RESOURCE_TYPE _Core3
  (* Standard: 61499-2 *)
  (* Version 0.1, 2017-00-16, hpea485, UOA *)
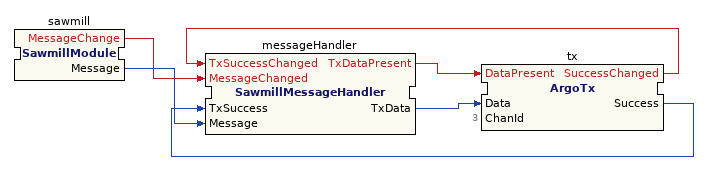
  FBS
    tx : ArgoTx(ChanId := 3);
    messageHandler : SawmillMessageHandler;
    sawmill : SawmillModule;
  END_FBS
  EVENT_CONNECTIONS
    tx.SuccessChanged TO messageHandler.TxSuccessChanged;
    messageHandler.TxDataPresent TO tx.DataPresent;
    sawmill.MessageChange TO messageHandler.MessageChanged;
  END_CONNECTIONS
  DATA_CONNECTIONS
    tx.Success TO messageHandler.TxSuccess;
    messageHandler.TxData TO tx.Data;
    sawmill.Message TO messageHandler.Message;
  END_CONNECTIONS
END_RESOURCE_TYPE
